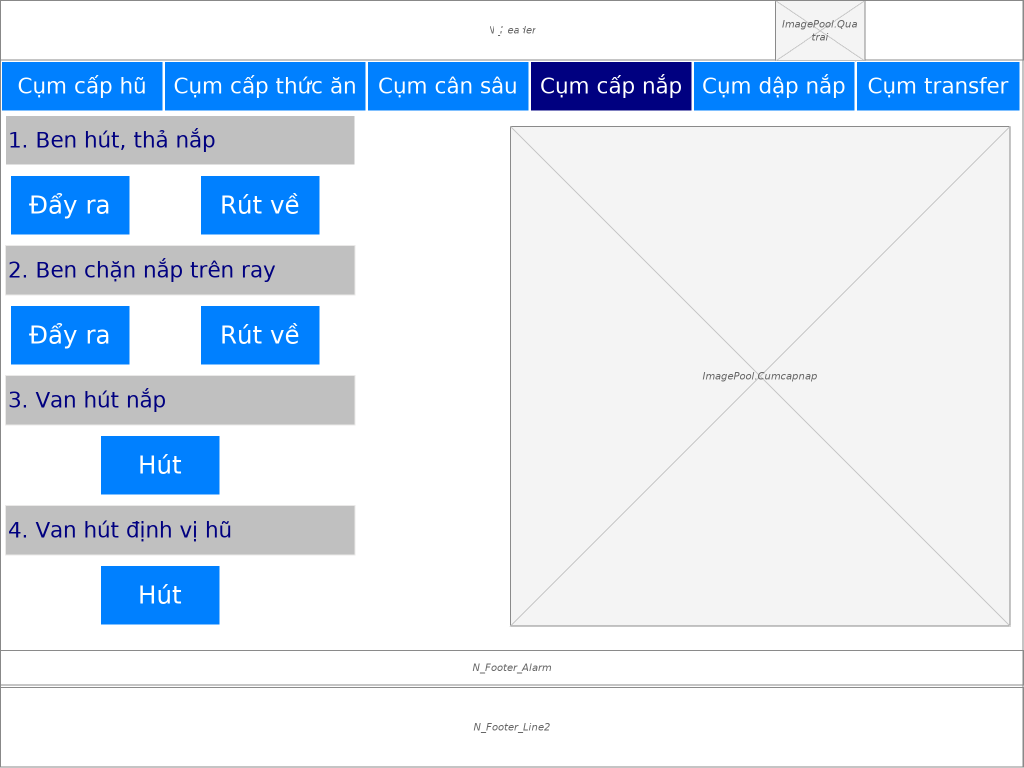
VISUALIZATION N_LidSupply2  // 1024x768
    Rectangle (10,305 120x60), "Đẩy ra", colour toggle: PR_Line02.bCylinder_LidStopper_extend
        OnMouseDown: execute { PR_Line02.bCylinder_LidStopper_extend := TRUE; PR_Line02.bCylinder_LidStopper_retract := FALSE; }
    Rectangle (200,175 120x60), "Rút về", colour toggle: PR_Line02.bCylinder_Suction_retract
        OnMouseDown: execute { PR_Line02.bCylinder_Suction_retract := TRUE; PR_Line02.bCylinder_Suction_extend := FALSE; }
    Rectangle (200,305 120x60), "Rút về", colour toggle: PR_Line02.bCylinder_LidStopper_retract
        OnMouseDown: execute { PR_Line02.bCylinder_LidStopper_retract := TRUE; PR_Line02.bCylinder_LidStopper_extend := FALSE; }
    Frame (0,687 1024x80)
        shows N_Footer_Line2()
    Frame (0,0 1024x60)
        shows N_Header()
    Textfield (353,5 400x50), "MÀN HÌNH CHẠY TAY LINE 2"
    Rectangle (10,175 120x60), "Đẩy ra", colour toggle: PR_Line02.bCylinder_Suction_extend
        OnMouseDown: execute { PR_Line02.bCylinder_Suction_extend := TRUE; PR_Line02.bCylinder_Suction_retract := FALSE; }
    Rectangle (100,435 120x60), "Dừng hút", invisible if: not PR_Line02.bLidSuctionValve, input disabled if: not PR_Line02.bLidSuctionValve
        OnMouseDown: execute { PR_Line02.bLidSuctionValve := FALSE; }
    Image (775,0 90x61), input disabled if: bResetAuto1, image: ImagePool.Qua trai
        OnMouseClick: change screen: N_LidSupply1
        OnMouseClick: execute { MAIN.bModeManual := TRUE; MAIN.bModeAuto := FALSE; }
    Rectangle (100,565 120x60), "Dừng hút", invisible if: not PR_Line02.bCupSuctionValve, input disabled if: not PR_Line02.bCupSuctionValve
        OnMouseDown: execute { PR_Line02.bCupSuctionValve := false; }
    Rectangle (1,61 162x50), "Cụm cấp hũ"
        OnMouseClick: change screen: N_JarSupply2
    Rectangle (164,61 202x50), "Cụm cấp thức ăn"
        OnMouseClick: change screen: N_FoodSupply2
    Rectangle (367,61 162x50), "Cụm cân sâu"
        OnMouseClick: change screen: N_WormWeight2
    Rectangle (530,61 162x50), "Cụm cấp nắp"
        OnMouseClick: change screen: N_LidSupply2
    Rectangle (693,61 162x50), "Cụm dập nắp"
        OnMouseClick: change screen: N_LidPressing2
    Rectangle (856,61 164x50), "Cụm transfer"
        OnMouseClick: change screen: N_Tranfer2
    Rectangle (100,435 120x60), "Hút", invisible if: PR_Line02.bLidSuctionValve, input disabled if: PR_Line02.bLidSuctionValve
        OnMouseDown: execute { PR_Line02.bLidSuctionValve := TRUE; }
    Rectangle (100,565 120x60), "Hút", invisible if: PR_Line02.bCupSuctionValve, input disabled if: PR_Line02.bCupSuctionValve
        OnMouseDown: execute { PR_Line02.bCupSuctionValve := true; }
    Image (510,126 500x500), image: ImagePool.Cumcapnap
    Rectangle (5,505 350x50), "4. Van hút định vị hũ"
    Rectangle (5,115 350x50), "1. Ben hút, thả nắp"
    Rectangle (5,245 350x50), "2. Ben chặn nắp trên ray"
    Rectangle (5,375 350x50), "3. Van hút nắp"
    Frame (0,650 1024x35)
        shows N_Footer_Alarm()
END_VISUALIZATION

(* stored: Version 1.1.0.1, ProductVersion 3.1.4024.12
   Visu N_LidSupply2: Id {340f5127-09a2-4241-bf18-f3657b18f2ad} *)
